// TIA Portal V20 export
DATA_BLOCK "idb_Conveyor_C3_DB"   // DB4
// stored: InstanceOfName C3.Conveyor_C3, InstanceOfType FB, Namespace C3
"C3.Conveyor_C3"
   // VAR
   //    R_TRIG_Instance { S7_SetPoint := 'True'} : R_TRIG;
   //    StatAutoRight { S7_SetPoint := 'True'} : Bool;
   // END_VAR
BEGIN
END_DATA_BLOCK
